Fanuc TP program (LS listing): S107_PK_T07N70.LS

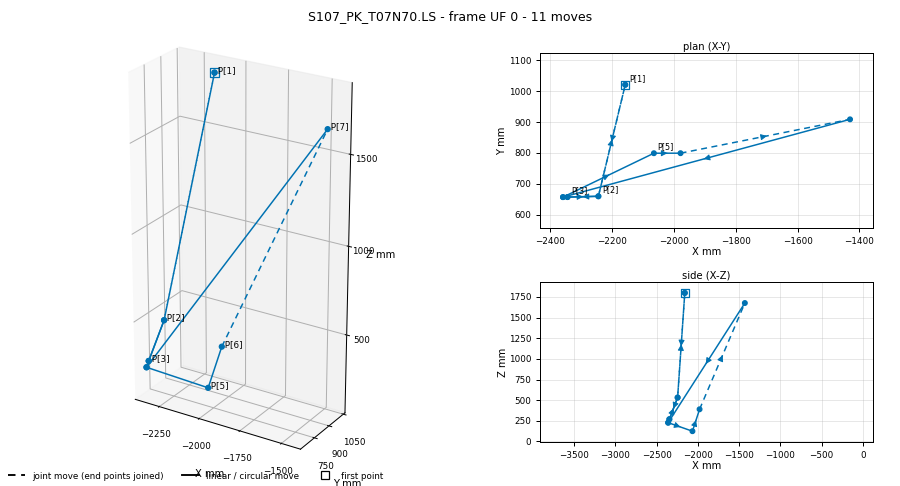
[picture p0: tool path of S107_PK_T07N70.LS in frame UF 0, 11 of 11 moves have a stored position in this frame; points joined in program order, loops and branches not executed]
/PROG  S107_PK_T07N70
/ATTR
OWNER		= MNEDITOR;
COMMENT		= "TL PCK TYP1 N70";
PROG_SIZE	= 4131;
CREATE		= DATE 18-11-03  TIME 14:37:36;
MODIFIED	= DATE 18-11-03  TIME 14:37:36;
FILE_NAME	= S001_PK_;
VERSION		= 0;
LINE_COUNT	= 151;
MEMORY_SIZE	= 4567;
PROTECT		= READ_WRITE;
STORAGE		= SHADOW;
TCD:  STACK_SIZE	= 0,
      TASK_PRIORITY	= 50,
      TIME_SLICE	= 0,
      BUSY_LAMP_OFF	= 0,
      ABORT_REQUEST	= 0,
      PAUSE_REQUEST	= 0;
DEFAULT_GROUP	= 1,*,*,*,*;
CONTROL_CODE	= 00000000 00000000;
/APPL
  HANDLING : TRUE ;
/MN
   1:  !******************************** ;
   2:  ! PATH - PK TOOL FROM N3=STA 70 ;
   3:  !******************************** ;
   4:  !* Robot ID: XXXXXR02B1 ;
   5:  !*    F-19XXXX ;
   6:  !* Line: XXXXXXXX ;
   7:  !* Platform: XX ;
   8:  !* Tool ID: TOOL xx ;
   9:  !* Program: S002_PK_TxxN3_R02 ;
  10:  !* Application: TOOL PICK ;
  11:  !******************************** ;
  12:  ! Author- Esys Automation ;
  13:  !******************************** ;
  14:   ;
  15:  !++++++++++++++++++++++++++++++++ ;
  16:  !ASSIGN PROGRAM PATH VALUES ;
  17:  !-------------------------------- ;
  18:  !Set ATI Tool and World UFrame ;
  19:  UTOOL_NUM=14 ;
  20:  UFRAME_NUM=0 ;
  21:  !++++++++++++++++++++++++++++++++ ;
  22:   ;
  23:  !******************************** ;
  24:  !BEGINNING OF PROGRAM PATH ;
  25:  !MOVE TO NEST 3 TOOL PICK ;
  26:  !******************************** ;
  27:   ;
  28:  !-------------------------------- ;
  29:  LBL[10:MOVE TO TL PICK] ;
  30:   ;
  31:  SET SEGMENT(52) ;
  32:  !SEG(52), Approach Tool Pick ;
  33:   ;
  34:J P[1] 100% CNT100    ;
  35:   ;
  36:J P[2:Tool-Pick-Pounce] 100% CNT100    ;
  37:   ;
  38:L P[3] 1000mm/sec CNT1    ;
  39:   ;
  40:L P[4:PICK_T07_N70] 50mm/sec FINE    ;
  41:   ;
  42:  !-------------------------------- ;
  43:  LBL[20:LATCH TOOL] ;
  44:  LATCH TOOL    ;
  45:   ;
  46:  !Add MH Ethernet Device from ;
  47:  !I/O Ethernet table ;
  48:  !which tool has ;
  49:   ;
  50:  !ADD DEVICE ONLINE CALLS ;
  51:  !WITHOUT STATUS CHECK ARG ;
  52:  !FOR ALL EOAT DEVICES ;
  53:  !CALL EN_ONLN(x,y) ;
  54:  !x = EOAT ENET Node # ;
  55:  !y = wait time ;
  56:  CALL EN_ONLN(31,5) ;
  57:  CALL EN_AROFF(31) ;
  58:   ;
  59:  !If TL LCH Pass, Return Home ;
  60:  !If TL LCH Fail, Unlatch TL, ;
  61:  !  MHFault, and Return Home ;
  62:  IF R[170]=1,JMP LBL[30] ;
  63:   ;
  64:  SELECT R[168]=6,JMP LBL[80] ;
  65:         ELSE,JMP LBL[99] ;
  66:   ;
  67:  !-------------------------------- ;
  68:  LBL[30:TOOL CHECK] ;
  69:   ;
  70:  ! Check if Tool Match with PLC ;
  71:  CALL TL_CHK_KM(R[156]) ;
  72:   ;
  73:  !If TL CHK Pass, Return Home ;
  74:  !If TL CHK Fail, Unlatch Tool, ;
  75:  !  MHFault, and Return Home ;
  76:  IF R[170]=1,JMP LBL[40] ;
  77:  IF R[170]=0,JMP LBL[905] ;
  78:   ;
  79:  !-------------------------------- ;
  80:  LBL[40:COMPLETE PATH] ;
  81:  !TL PK COMPLETE. MOVE AWAY ;
  82:  !AND RETURN HOME ;
  83:   ;
  84:  !Set New Tool and World Frame ;
  85:  UTOOL_NUM=2 ;
  86:  UFRAME_NUM=0 ;
  87:   ;
  88:  !Set Payload= Tool ;
  89:  R[221]=2    ;
  90:  PAYLOAD[R[221]] ;
  91:   ;
  92:  SET SEGMENT(53) ;
  93:  !SEG(53), Tool Pick Depart ;
  94:   ;
  95:L P[5] 50mm/sec FINE    ;
  96:L P[6] 1000mm/sec CNT50    ;
  97:   ;
  98:J P[7] 100% CNT100    ;
  99:   ;
 100:  ! Move To Home ;
 101:  JMP LBL[100] ;
 102:   ;
 103:  !-------------------------------- ;
 104:  LBL[80:LATCHING FAULT] ;
 105:  !MOVE BACK TO HOME WITHOUT TOOL ;
 106:  !on Reverse Path before Tool Pick ;
 107:   ;
 108:  UNLATCH TOOL    ;
 109:   ;
 110:  UFRAME_NUM=0 ;
 111:  UTOOL_NUM=14 ;
 112:   ;
 113:L P[4:PICK_T07_N70] 50mm/sec FINE    ;
 114:L P[3] 500mm/sec FINE    ;
 115:   ;
 116:L P[2:Tool-Pick-Pounce] 750mm/sec CNT100    ;
 117:   ;
 118:J P[1] 100% CNT100    ;
 119:   ;
 120:  SET SEGMENT(63) ;
 121:  !SEG(63), Robot Move to Home ;
 122:   ;
 123:  R[132]=0    ;
 124:  GO[71]=0 ;
 125:   ;
 126:  ! Move To Home ;
 127:  JMP LBL[100] ;
 128:   ;
 129:  !-------------------------------- ;
 130:  LBL[99:ABORT PROGRAM] ;
 131:  MESSAGE[...] ;
 132:  MESSAGE[ABORT PROGRAM] ;
 133:  ABORT ;
 134:   ;
 135:  !-------------------------------- ;
 136:  LBL[100:END OF PROGRAM] ;
 137:  END ;
 138:   ;
 139:  !***********FAULTS*********** ;
 140:  LBL[905:Invalid Tool Num] ;
 141:  MESSAGE[...] ;
 142:  MESSAGE[TOOL CHANGER FAULT] ;
 143:  MESSAGE[ ROBOT LATCHED TO] ;
 144:  MESSAGE[ WRONG TOOL.] ;
 145:  MESSAGE[ GI[70] DOES NOT ] ;
 146:  MESSAGE[ MATCH TOOL ID ] ;
 147:  DO[523]=ON ;
 148:  UALM[3] ;
 149:  DO[523]=OFF ;
 150:  JMP LBL[80] ;
 151:   ;
/POS
P[1]{
   GP1:
	UF : 0, UT : 14,		CONFIG : 'N U T, 0, 0, 0',
	X = -2157.965  mm,	Y =  1020.774  mm,	Z =  1799.157  mm,
	W =  -148.691 deg,	P =     -.556 deg,	R =    64.095 deg
};
P[2:"Tool-Pick-Pounce"]{
   GP1:
	UF : 0, UT : 14,		CONFIG : 'N U T, 0, 0, 0',
	X = -2244.914  mm,	Y =   659.821  mm,	Z =   531.956  mm,
	W =  -159.212 deg,	P =      .429 deg,	R =    91.141 deg
};
P[3]{
   GP1:
	UF : 0, UT : 14,		CONFIG : 'N U T, 0, 0, 0',
	X = -2344.885  mm,	Y =   657.166  mm,	Z =   269.226  mm,
	W =  -160.469 deg,	P =     -.183 deg,	R =    90.925 deg
};
P[4:"PICK_T07_N70"]{
   GP1:
	UF : 0, UT : 14,		CONFIG : 'N U T, 0, 0, 0',
	X = -2359.541  mm,	Y =   657.062  mm,	Z =   227.911  mm,
	W =  -160.469 deg,	P =     -.183 deg,	R =    90.925 deg
};
P[5]{
   GP1:
	UF : 0, UT : 2,		CONFIG : 'N U T, 0, 0, 0',
	X = -2065.274  mm,	Y =   799.180  mm,	Z =   124.447  mm,
	W =  -162.006 deg,	P =      .170 deg,	R =    89.547 deg
};
P[6]{
   GP1:
	UF : 0, UT : 2,		CONFIG : 'N U T, 0, 0, 0',
	X = -1979.057  mm,	Y =   799.286  mm,	Z =   389.879  mm,
	W =  -162.006 deg,	P =      .170 deg,	R =    89.547 deg
};
P[7]{
   GP1:
	UF : 0, UT : 2,		CONFIG : 'N U T, 0, 0, 0',
	X = -1430.516  mm,	Y =   908.811  mm,	Z =  1676.906  mm,
	W =  -145.907 deg,	P =     1.406 deg,	R =    88.198 deg
};
/END
